// TIA Portal V20 export
FUNCTION "纠偏伺服" : Void   // FC1, LAD
{ S7_Optimized_Access := 'TRUE' }
// stored: SetENOAutomatically false
BEGIN

REGION Network 1 (SCL)
   "纠偏V90控制字".%X0:="G2_下载".位1;
   "纠偏V90控制字".%X1 := "G2_下载".位2;
   "纠偏V90控制字".%X2 := "G2_下载".位3;
   "纠偏V90控制字".%X3 := "G2_下载".位4;
   "纠偏V90控制字".%X4 := "G2_下载".位5;
   "纠偏V90控制字".%X5 := "G2_下载".位6;
   "纠偏V90控制字".%X6 := "G2_下载".位7;
   "纠偏V90控制字".%X7 := "G2_下载".位8;

   "纠_回原模式" := "G2_下载".整型1;

   "纠_绝对位置" := "G2_下载".浮点数1;
   "纠_绝对速度" := "G2_下载".浮点数2;
   "纠_相对位置" := "G2_下载".浮点数3;
   "纠_相对位置" := "G2_下载".浮点数4;
   "纠_点动速度" := "G2_下载".浮点数5;
END_REGION

REGION Network 2
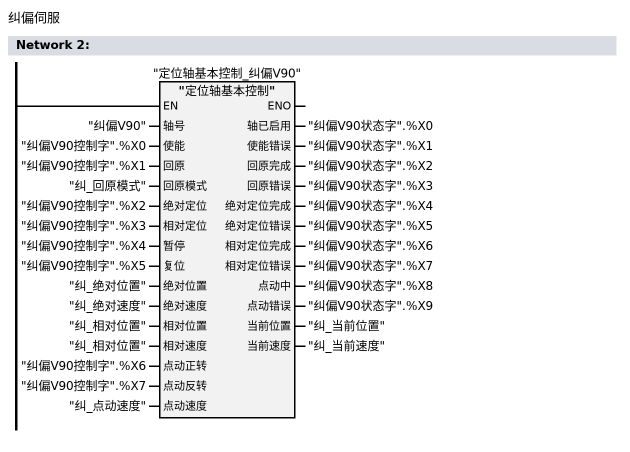
   RUNG wire#powerrail
      "定位轴基本控制_纠偏V90"(轴号 := "纠偏V90", 使能 := "纠偏V90控制字".%X0, 回原 := "纠偏V90控制字".%X1, 回原模式 := "纠_回原模式", 绝对定位 := "纠偏V90控制字".%X2, 相对定位 := "纠偏V90控制字".%X3, 暂停 := "纠偏V90控制字".%X4, 复位 := "纠偏V90控制字".%X5, 绝对位置 := "纠_绝对位置", 绝对速度 := "纠_绝对速度", 相对位置 := "纠_相对位置", 相对速度 := "纠_相对位置", 点动正转 := "纠偏V90控制字".%X6, 点动反转 := "纠偏V90控制字".%X7, 点动速度 := "纠_点动速度", 轴已启用 => "纠偏V90状态字".%X0, 使能错误 => "纠偏V90状态字".%X1, 回原完成 => "纠偏V90状态字".%X2, 回原错误 => "纠偏V90状态字".%X3, 绝对定位完成 => "纠偏V90状态字".%X4, 绝对定位错误 => "纠偏V90状态字".%X5, 相对定位完成 => "纠偏V90状态字".%X6, 相对定位错误 => "纠偏V90状态字".%X7, 点动中 => "纠偏V90状态字".%X8, 点动错误 => "纠偏V90状态字".%X9, 当前位置 => "纠_当前位置", 当前速度 => "纠_当前速度")
   END_RUNG
   // the same network as SCL:
   "定位轴基本控制_纠偏V90"(轴号 := "纠偏V90",   // "定位轴基本控制"
                   使能 := "纠偏V90控制字".%X0,
                   回原 := "纠偏V90控制字".%X1,
                   回原模式 := "纠_回原模式",
                   绝对定位 := "纠偏V90控制字".%X2,
                   相对定位 := "纠偏V90控制字".%X3,
                   暂停 := "纠偏V90控制字".%X4,
                   复位 := "纠偏V90控制字".%X5,
                   绝对位置 := "纠_绝对位置",
                   绝对速度 := "纠_绝对速度",
                   相对位置 := "纠_相对位置",
                   相对速度 := "纠_相对位置",
                   点动正转 := "纠偏V90控制字".%X6,
                   点动反转 := "纠偏V90控制字".%X7,
                   点动速度 := "纠_点动速度",
                   轴已启用 => "纠偏V90状态字".%X0,
                   使能错误 => "纠偏V90状态字".%X1,
                   回原完成 => "纠偏V90状态字".%X2,
                   回原错误 => "纠偏V90状态字".%X3,
                   绝对定位完成 => "纠偏V90状态字".%X4,
                   绝对定位错误 => "纠偏V90状态字".%X5,
                   相对定位完成 => "纠偏V90状态字".%X6,
                   相对定位错误 => "纠偏V90状态字".%X7,
                   点动中 => "纠偏V90状态字".%X8,
                   点动错误 => "纠偏V90状态字".%X9,
                   当前位置 => "纠_当前位置",
                   当前速度 => "纠_当前速度");
END_REGION

REGION Network 3 (SCL)
   "G2_上传".位1 := "纠偏V90状态字".%X0;
   "G2_上传".位2 := "纠偏V90状态字".%X1;
   "G2_上传".位3 := "纠偏V90状态字".%X2;
   "G2_上传".位4 := "纠偏V90状态字".%X3;
   "G2_上传".位5 := "纠偏V90状态字".%X4;
   "G2_上传".位6 := "纠偏V90状态字".%X5;
   "G2_上传".位7 := "纠偏V90状态字".%X6;
   "G2_上传".位8 := "纠偏V90状态字".%X7;
   "G2_上传".位9 := "纠偏V90状态字".%X8;
   "G2_上传".位10 := "纠偏V90状态字".%X9;

   "G2_上传".浮点数1 := LREAL_TO_REAL(IN := "纠_当前位置");
   "G2_上传".浮点数2 := LREAL_TO_REAL(IN := "纠_当前速度");
END_REGION
END_FUNCTION
